FUNCTION_BLOCK FB_Rpc
VAR_INPUT
END_VAR
VAR_OUTPUT
END_VAR
VAR
END_VAR

{attribute 'TcRpcEnable'}
METHOD Calculator : BOOL
VAR_INPUT
	Value1	: REAL;
	Value2	: REAL;
END_VAR
VAR_OUTPUT
	Sum			: REAL;
	Product 	: REAL;
	Division	: REAL;
END_VAR
//Return TRUE if all success
Calculator := TRUE;

Sum := Value1 + Value2;
Product := Value1 * Value2;

IF Value2 <> 0 THEN
	Division := Value1 / Value2;
ELSE
	Division := 0;
	Calculator := FALSE;
END_IF
END_METHOD

{attribute 'TcRpcEnable'}
METHOD StructTest : ST_Struct
VAR_INPUT
	Input	: ST_Struct;
END_VAR
StructTest.SomeText := CONCAT('Response: ', Input.SomeText);
StructTest.SomeReal := Input.SomeReal * 10.0;
StructTest.SomeDate := Input.SomeDate + T#24H;
END_METHOD

END_FUNCTION_BLOCK

(* stored: Version 1.1.0.1, ProductVersion 3.1.4024.12
   POU FB_Rpc: Id {85a5d823-5c41-4c26-a181-82a08e3d478f}, SpecialFunc None
   Method Calculator: Id {f0891cd6-229e-4300-8553-fa06a430c8f0}
   Method StructTest: Id {6ef4d474-76c0-4d34-920e-b9c2c4860978} *)
